{attribute 'GeneratedUsingTerminal: EP2316-0003-0016'}
{attribute addProperty BoxType "EP2316-0003-0016"}
{attribute addProperty Id "Diag_InputAT %I*ARRAY[0..7] OF BOOL8"}
{attribute addProperty CRC "568896300"}
{attribute addProperty Size "8"}
TYPE DIG_Diag_Inputs_584303BF :
STRUCT
	{attribute addProperty Name "Diag_Input"}
	Diag_Input AT %I* : ARRAY[0..7] OF BOOL;
END_STRUCT
END_TYPE

(* stored: Version 1.2.0.0, ProductVersion 3.1.4024.9
   DUT DIG_Diag_Inputs_584303BF: Id {bb291b24-d242-4f11-81ad-aa95e34ac4e2} *)
